(* CODESYS project 2019-30-07-Sparkplug_Publish.ecp

Project tree, tasks and I/O mapping:
  PFC_Sparkplug : 750-8212 PFC200 2ETH RS, WAGO, order no. 0750-8212, version 5.13.2.32
    application Application
      libraries: CIP Encapsulation Layer, 3.5.13.0 (3S - Smart Software Solutions GmbH); WagoAppJSON, 1.0.2.0 (WAGO); WagoAppCloud, * (WAGO)
      task PLC_Task (cyclic, interval t#50ms, priority 15) calls PLC_PRG
      program PLC_PRG [ST]
      program VariableLoggerCyclic [ST]
      program VariableLoggerEvent [ST]
    Kbus : Kbus, WAGO, version 1.4.0.2
        unmapped channels: K-BUS diagnostics
    MODBUS
      MODBUS : MODBUS, WAGO, order no. n/a, version 1.1.1.15
    Common.PCI
    Serial
      COM1 : COM1, WAGO, version 0.0.0.19
*)

// PFC_Sparkplug/Application/PLC_PRG
PROGRAM PLC_PRG
VAR
	simu: BOOL := 0;		
	levelTank1:INT:=0;
	levelTank2:INT:=0;
	levelTank3:INT:=0;
END_VAR



//VariableLoggerCyclic(levelTank1:=actLevelTank1,levelTank2:=actLevelTank2,levelTank3:=actLevelTank3);
VariableLoggerEvent(switchState:=simu, levelTank1:=levelTank1,levelTank2:=levelTank2,levelTank3:=levelTank3);

END_PROGRAM

// PFC_Sparkplug/Application/VariableLoggerCyclic
PROGRAM VariableLoggerCyclic
VAR_INPUT
	levelTank1: INT := 0;
	levelTank2: INT := 0;
	levelTank3: INT := 0;
END_VAR
VAR RETAIN
	/// Remanent variables 
	tSampleInterval1: TIME := TIME#10s0ms;
	tPublishInterval1: TIME := TIME#10s0ms;
END_VAR
VAR
	/// Define one collection
	aCollections: ARRAY[0..0] OF WagoAppCloud.typCollection;
	/// Define 3 variables for the collection
	aVariableDescriptions1: ARRAY[0..2] OF WagoAppCloud.typVariableDescription;
	oFbCollectionLogger: WagoAppCloud.FbCollectionLogger;
END_VAR

(* Init collection 1 *)
aVariableDescriptions1[0].pAddress := ADR(levelTank1);
aVariableDescriptions1[0].eValueType := WagoAppCloud.VVT_INT;
aVariableDescriptions1[0].dwTypeId := 1;
aVariableDescriptions1[0].sTag := 'Tank_1';
aVariableDescriptions1[0].sUnit := '%';

aVariableDescriptions1[1].pAddress := ADR(levelTank2);
aVariableDescriptions1[1].eValueType := WagoAppCloud.VVT_INT;
aVariableDescriptions1[1].dwTypeId := 2;
aVariableDescriptions1[1].sTag := 'Tank_2';
aVariableDescriptions1[1].sUnit := '%';

aVariableDescriptions1[2].pAddress := ADR(levelTank3);
aVariableDescriptions1[2].eValueType := WagoAppCloud.VVT_INT;
aVariableDescriptions1[2].dwTypeId := 3;
aVariableDescriptions1[2].sTag := 'Tank_3';
aVariableDescriptions1[2].sUnit := '%';

aCollections[0].dwCollectionId := 1;
aCollections[0].sName := 'Collection1';
aCollections[0].pSampleInterval := ADR(tSampleInterval1);
aCollections[0].pPublishInterval := ADR(tPublishInterval1);
aCollections[0].pVariableDescriptions := ADR(aVariableDescriptions1);
aCollections[0].dwVariablesCount := 3;

oFbCollectionLogger(pCollections := ADR(aCollections),
					dwCollectionsCount := 1);

END_PROGRAM

// PFC_Sparkplug/Application/VariableLoggerEvent
PROGRAM VariableLoggerEvent
VAR_INPUT
	switchState: BOOL := FALSE;
	levelTank1: INT := 0;
	levelTank2: INT := 0;
	levelTank3: INT := 0;
END_VAR
VAR RETAIN
	/// Remanent variables 
	tPublishInterval1: TIME := TIME#0ms;	// due to publish on value change 0 
END_VAR
VAR
	/// Define one collection
	aCollections: ARRAY[0..0] OF WagoAppCloud.typCollection;
	/// Define 4 variables for the collection
	aVariableDescriptions1: ARRAY[0..3] OF WagoAppCloud.typVariableDescription;
	oFbCollectionLogger: WagoAppCloud.FbCollectionLogger;
	oldLevelTank1: INT := 0;
	oldLevelTank2: INT := 0;
	oldLevelTank3: INT := 0;
	oldSwitchState: BOOL := FALSE;
END_VAR

// set trigger of variables on value change 
IF (levelTank1 <> oldLevelTank1) THEN
	oldLevelTank1 := levelTank1;
	aVariableDescriptions1[0].xVariableTrigger:=TRUE;
ELSE
	aVariableDescriptions1[0].xVariableTrigger:=FALSE;
END_IF

IF (levelTank2 <> oldLevelTank2) THEN
	oldLevelTank2 := levelTank2;
	aVariableDescriptions1[1].xVariableTrigger:=TRUE;
ELSE
	aVariableDescriptions1[1].xVariableTrigger:=FALSE;
END_IF

IF (levelTank3 <> oldLevelTank3) THEN
	oldLevelTank3 := levelTank3;
	aVariableDescriptions1[2].xVariableTrigger:=TRUE;
ELSE
	aVariableDescriptions1[2].xVariableTrigger:=FALSE;
END_IF

IF (SwitchState <> oldSwitchState) THEN
	oldSwitchState := SwitchState;
	aVariableDescriptions1[3].xVariableTrigger:=TRUE;
ELSE
	aVariableDescriptions1[3].xVariableTrigger:=FALSE;
END_IF

(* Init collection 1 *)
aVariableDescriptions1[0].pAddress := ADR(levelTank1);
aVariableDescriptions1[0].eValueType := WagoAppCloud.VVT_INT;
aVariableDescriptions1[0].dwTypeId := 1;
aVariableDescriptions1[0].sTag := 'Tank_1';
aVariableDescriptions1[0].sUnit := '%';

aVariableDescriptions1[1].pAddress := ADR(levelTank2);
aVariableDescriptions1[1].eValueType := WagoAppCloud.VVT_INT;
aVariableDescriptions1[1].dwTypeId := 2;
aVariableDescriptions1[1].sTag := 'Tank_2';
aVariableDescriptions1[1].sUnit := '%';

aVariableDescriptions1[2].pAddress := ADR(levelTank3);
aVariableDescriptions1[2].eValueType := WagoAppCloud.VVT_INT;
aVariableDescriptions1[2].dwTypeId := 3;
aVariableDescriptions1[2].sTag := 'Tank_3';
aVariableDescriptions1[2].sUnit := '%';

aVariableDescriptions1[3].pAddress := ADR(switchState);
aVariableDescriptions1[3].eValueType := WagoAppCloud.VVT_BOOL;
aVariableDescriptions1[3].dwTypeId := 4;
aVariableDescriptions1[3].sTag := 'State';
aVariableDescriptions1[3].sUnit := '';

aCollections[0].dwCollectionId := 1;
aCollections[0].sName := 'Collection1';
aCollections[0].pPublishInterval := ADR(tPublishInterval1);
aCollections[0].pVariableDescriptions := ADR(aVariableDescriptions1);
aCollections[0].dwVariablesCount := 4;
aCollections[0].eSamplingDataMode := eSamplingMode.UNEQUALLY_SPACED_CUSTOMIZED_SAMPLES;

oFbCollectionLogger(pCollections := ADR(aCollections),
					dwCollectionsCount := 1);

END_PROGRAM
